(*

short summary
=============
A specialized candy. It can be consumed by any candy consumer.
It supports dynamic creation. Furthermore, it calls the method 
AbstractCandy.initializeDispatchers after FB_init.

legal notes
===========
SPDX-FileCopyrightText: © 2024 ekvip automation GmbH <info@ekvip.de>
SPDX-License-Identifier: Apache-2.0
For details check: Apache-2.0_

.. _Apache-2.0: https://www.apache.org/licenses/LICENSE-2.0

*)

{attribute 'enable_dynamic_creation'}
{attribute 'call_after_init'}
FUNCTION_BLOCK FINAL Altoids EXTENDS AbstractCandy
VAR_INPUT
END_VAR
VAR_OUTPUT
END_VAR
VAR
END_VAR

(*

short summary
=============
it initializes the amount, the candy name and 
the binary coded candy type  

legal notes
===========
SPDX-FileCopyrightText: © 2024 ekvip automation GmbH <info@ekvip.de>
SPDX-License-Identifier: Apache-2.0
For details check: Apache-2.0_

.. _Apache-2.0: https://www.apache.org/licenses/LICENSE-2.0

*)

METHOD FB_init :BOOL
VAR_INPUT
	(* if TRUE, the retain variables are initialized (warm start / cold start) *)
	bInitRetains	:BOOL;
	(* if TRUE, the instance afterwards gets moved into the copy code (online change) *)
	bInCopyCode		:BOOL;
END_VAR
THIS^.amount := 50;
THIS^.name := 'Altoids Classic Peppermint';
THIS^.candyType := CandyTypes.MINTS;
END_METHOD

END_FUNCTION_BLOCK

(* stored: Version 1.1.0.1
   POU Altoids: Id {5412c823-aea5-45d1-aff0-e8fd503ca3c3}, SpecialFunc None
   Method FB_init: Id {b7851a9f-5884-4560-beae-2a20d1ac2afa} *)
